{attribute 'qualified_only'}
{attribute 'strict'}
{attribute 'to_string'}
TYPE E_RecipeStepCommand :
(
	Idle := 0,
	Heat,
	Cool,
	Mix,
	Pump
)BYTE;
END_TYPE

(* stored: Version 1.1.0.1, ProductVersion 3.1.4024.15
   EnumerationTextList E_RecipeStepCommand: Id {65e45cd4-aa7d-4f01-b110-3d623c02e4b4} *)
